// TIA Portal V17 export
// export: Created 2023-09-11T16:36:44.884775Z, ExportSetting WithDefaults, DisplayName Totally Integrated Automation Portal, DisplayVersion V17 Update 6, DisplayName TIA Portal Openness, DisplayVersion V17 Update 6, DisplayName TIA Portal Teamcenter Gateway, DisplayVersion V17 Update 6, DisplayName TIA Portal Version Control Interface, DisplayVersion V17, DisplayName Simotion SCOUT TIA, DisplayVersion 5.4.3.0, DisplayName TIA Portal Test Suite Advanced, DisplayVersion V17 Update 1, DisplayName SIMOCODE ES, DisplayVersion V17 Update 5, DisplayName SINAMICS Startdrive Advanced, DisplayVersion V17 SP1, DisplayName SINAMICS Startdrive G130, G150, S120, S150, SINAMICS MV, S210, DisplayVersion V17 SP1, DisplayName SINAMICS Startdrive G110M, G120, G120C, G120D, G120P, G115D, DisplayVersion V17 SP1, DisplayName SIRIUS Safety ES, DisplayVersion V17 Update 5, DisplayName STEP 7 Professional, DisplayVersion V17 Update 6, DisplayName STEP 7 CFC, DisplayVersion V17 Update 1, DisplayName STEP 7 Safety, DisplayVersion V17 Update 6, DisplayName WinCC Advanced, DisplayVersion V17 Update 6, DisplayName SIMATIC Visualization Architect, DisplayVersion V17 Update 5
FUNCTION "08_Gate Manager" : Void   // FC9, F_LAD
{ S7_Optimized_Access := 'TRUE' }
VERSION : 0.1
// stored: AutoNumber true, IsIECCheckEnabled false, UDAEnableTagReadback false
   VAR_TEMP
      temp_EXAMPLE_OPEN : Bool;
   END_VAR
BEGIN

REGION Network 1: S1 - SE01-B1 ([D002] P1004 | =SC01+LV004.EL001/310)
   // Sorter Gate
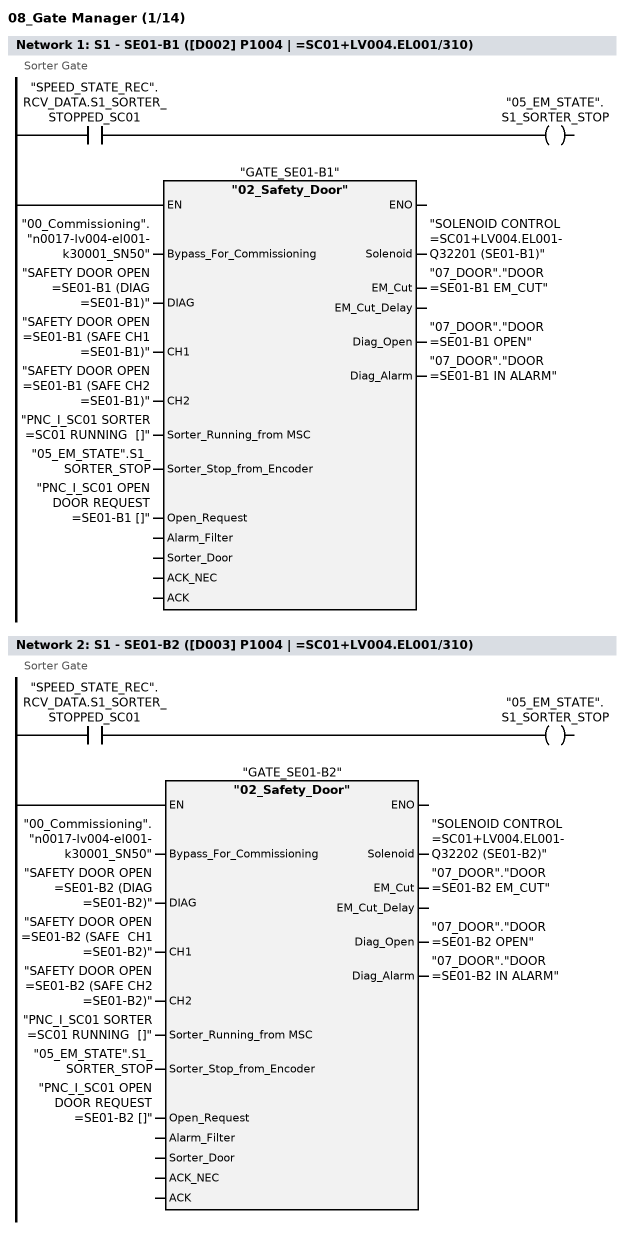
   RUNG wire#powerrail
      Contact( "SPEED_STATE_REC".RCV_DATA.S1_SORTER_STOPPED_SC01 )
      Coil( "05_EM_STATE".S1_SORTER_STOP )
   END_RUNG
   RUNG wire#powerrail
      "GATE_SE01-B1"(Bypass_For_Commissioning := "00_Commissioning"."n0017-lv004-el001-k30001_SN50", DIAG := "SAFETY DOOR OPEN =SE01-B1 (DIAG  =SE01-B1)", CH1 := "SAFETY DOOR OPEN =SE01-B1 (SAFE CH1 =SE01-B1)", CH2 := "SAFETY DOOR OPEN =SE01-B1 (SAFE CH2 =SE01-B1)", "Sorter_Running_from MSC" := "PNC_I_SC01 SORTER =SC01 RUNNING  []", Sorter_Stop_from_Encoder := "05_EM_STATE".S1_SORTER_STOP, Open_Request := "PNC_I_SC01 OPEN DOOR REQUEST =SE01-B1 []", Alarm_Filter :=, Sorter_Door :=, ACK_NEC :=, ACK :=, Solenoid => "SOLENOID CONTROL =SC01+LV004.EL001-Q32201 (SE01-B1)", EM_Cut => "07_DOOR"."DOOR =SE01-B1 EM_CUT", EM_Cut_Delay =>, Diag_Open => "07_DOOR"."DOOR =SE01-B1 OPEN", Diag_Alarm => "07_DOOR"."DOOR =SE01-B1 IN ALARM")
   END_RUNG
   // the same network as SCL:
   "05_EM_STATE".S1_SORTER_STOP := "SPEED_STATE_REC".RCV_DATA.S1_SORTER_STOPPED_SC01;
   "GATE_SE01-B1"(Bypass_For_Commissioning := "00_Commissioning"."n0017-lv004-el001-k30001_SN50",   // "02_Safety_Door"
                  DIAG := "SAFETY DOOR OPEN =SE01-B1 (DIAG  =SE01-B1)",
                  CH1 := "SAFETY DOOR OPEN =SE01-B1 (SAFE CH1 =SE01-B1)",
                  CH2 := "SAFETY DOOR OPEN =SE01-B1 (SAFE CH2 =SE01-B1)",
                  "Sorter_Running_from MSC" := "PNC_I_SC01 SORTER =SC01 RUNNING  []",
                  Sorter_Stop_from_Encoder := "05_EM_STATE".S1_SORTER_STOP,
                  Open_Request := "PNC_I_SC01 OPEN DOOR REQUEST =SE01-B1 []",
                  Solenoid => "SOLENOID CONTROL =SC01+LV004.EL001-Q32201 (SE01-B1)",
                  EM_Cut => "07_DOOR"."DOOR =SE01-B1 EM_CUT",
                  Diag_Open => "07_DOOR"."DOOR =SE01-B1 OPEN",
                  Diag_Alarm => "07_DOOR"."DOOR =SE01-B1 IN ALARM");
END_REGION

REGION Network 2: S1 - SE01-B2 ([D003] P1004 | =SC01+LV004.EL001/310)
   // Sorter Gate
   RUNG wire#powerrail
      Contact( "SPEED_STATE_REC".RCV_DATA.S1_SORTER_STOPPED_SC01 )
      Coil( "05_EM_STATE".S1_SORTER_STOP )
   END_RUNG
   RUNG wire#powerrail
      "GATE_SE01-B2"(Bypass_For_Commissioning := "00_Commissioning"."n0017-lv004-el001-k30001_SN50", DIAG := "SAFETY DOOR OPEN =SE01-B2 (DIAG  =SE01-B2)", CH1 := "SAFETY DOOR OPEN =SE01-B2 (SAFE  CH1 =SE01-B2)", CH2 := "SAFETY DOOR OPEN =SE01-B2 (SAFE CH2 =SE01-B2)", "Sorter_Running_from MSC" := "PNC_I_SC01 SORTER =SC01 RUNNING  []", Sorter_Stop_from_Encoder := "05_EM_STATE".S1_SORTER_STOP, Open_Request := "PNC_I_SC01 OPEN DOOR REQUEST =SE01-B2 []", Alarm_Filter :=, Sorter_Door :=, ACK_NEC :=, ACK :=, Solenoid => "SOLENOID CONTROL =SC01+LV004.EL001-Q32202 (SE01-B2)", EM_Cut => "07_DOOR"."DOOR =SE01-B2 EM_CUT", EM_Cut_Delay =>, Diag_Open => "07_DOOR"."DOOR =SE01-B2 OPEN", Diag_Alarm => "07_DOOR"."DOOR =SE01-B2 IN ALARM")
   END_RUNG
   // the same network as SCL:
   "05_EM_STATE".S1_SORTER_STOP := "SPEED_STATE_REC".RCV_DATA.S1_SORTER_STOPPED_SC01;
   "GATE_SE01-B2"(Bypass_For_Commissioning := "00_Commissioning"."n0017-lv004-el001-k30001_SN50",   // "02_Safety_Door"
                  DIAG := "SAFETY DOOR OPEN =SE01-B2 (DIAG  =SE01-B2)",
                  CH1 := "SAFETY DOOR OPEN =SE01-B2 (SAFE  CH1 =SE01-B2)",
                  CH2 := "SAFETY DOOR OPEN =SE01-B2 (SAFE CH2 =SE01-B2)",
                  "Sorter_Running_from MSC" := "PNC_I_SC01 SORTER =SC01 RUNNING  []",
                  Sorter_Stop_from_Encoder := "05_EM_STATE".S1_SORTER_STOP,
                  Open_Request := "PNC_I_SC01 OPEN DOOR REQUEST =SE01-B2 []",
                  Solenoid => "SOLENOID CONTROL =SC01+LV004.EL001-Q32202 (SE01-B2)",
                  EM_Cut => "07_DOOR"."DOOR =SE01-B2 EM_CUT",
                  Diag_Open => "07_DOOR"."DOOR =SE01-B2 OPEN",
                  Diag_Alarm => "07_DOOR"."DOOR =SE01-B2 IN ALARM");
END_REGION

REGION Network 3: S1 - SE01-B3 ([D012] F1001 | =SC01+MA001.EL001/310)
   // Sorter Gate
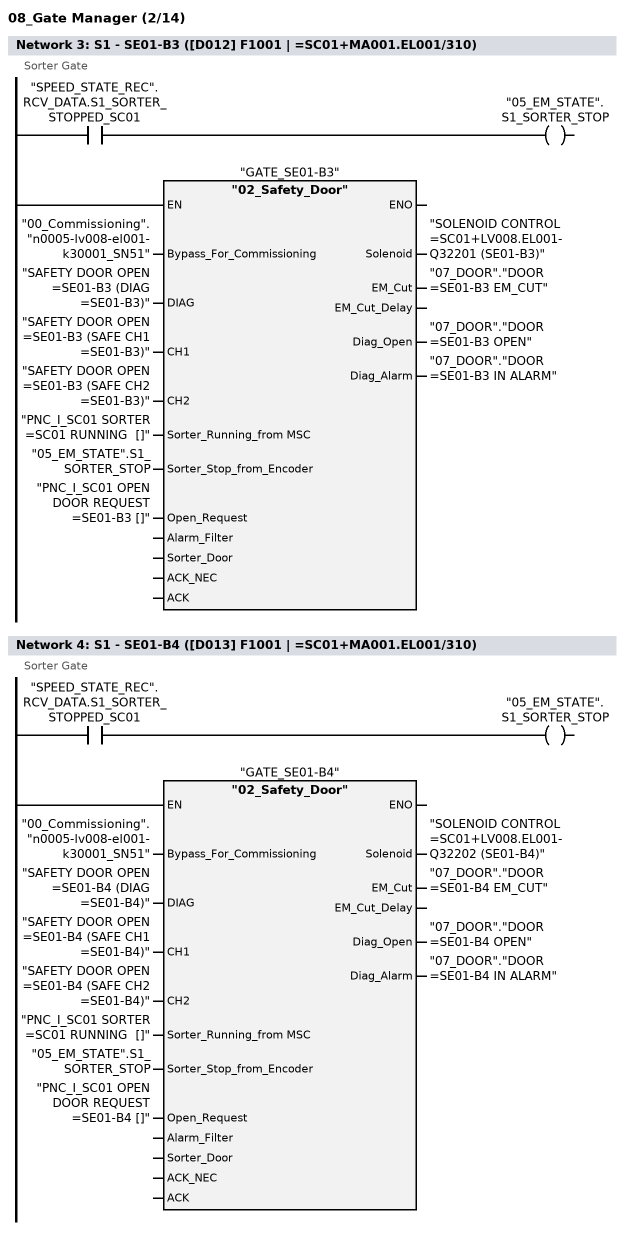
   RUNG wire#powerrail
      Contact( "SPEED_STATE_REC".RCV_DATA.S1_SORTER_STOPPED_SC01 )
      Coil( "05_EM_STATE".S1_SORTER_STOP )
   END_RUNG
   RUNG wire#powerrail
      "GATE_SE01-B3"(Bypass_For_Commissioning := "00_Commissioning"."n0005-lv008-el001-k30001_SN51", DIAG := "SAFETY DOOR OPEN =SE01-B3 (DIAG =SE01-B3)", CH1 := "SAFETY DOOR OPEN =SE01-B3 (SAFE CH1 =SE01-B3)", CH2 := "SAFETY DOOR OPEN =SE01-B3 (SAFE CH2 =SE01-B3)", "Sorter_Running_from MSC" := "PNC_I_SC01 SORTER =SC01 RUNNING  []", Sorter_Stop_from_Encoder := "05_EM_STATE".S1_SORTER_STOP, Open_Request := "PNC_I_SC01 OPEN DOOR REQUEST =SE01-B3 []", Alarm_Filter :=, Sorter_Door :=, ACK_NEC :=, ACK :=, Solenoid => "SOLENOID CONTROL =SC01+LV008.EL001-Q32201 (SE01-B3)", EM_Cut => "07_DOOR"."DOOR =SE01-B3 EM_CUT", EM_Cut_Delay =>, Diag_Open => "07_DOOR"."DOOR =SE01-B3 OPEN", Diag_Alarm => "07_DOOR"."DOOR =SE01-B3 IN ALARM")
   END_RUNG
   // the same network as SCL:
   "05_EM_STATE".S1_SORTER_STOP := "SPEED_STATE_REC".RCV_DATA.S1_SORTER_STOPPED_SC01;
   "GATE_SE01-B3"(Bypass_For_Commissioning := "00_Commissioning"."n0005-lv008-el001-k30001_SN51",   // "02_Safety_Door"
                  DIAG := "SAFETY DOOR OPEN =SE01-B3 (DIAG =SE01-B3)",
                  CH1 := "SAFETY DOOR OPEN =SE01-B3 (SAFE CH1 =SE01-B3)",
                  CH2 := "SAFETY DOOR OPEN =SE01-B3 (SAFE CH2 =SE01-B3)",
                  "Sorter_Running_from MSC" := "PNC_I_SC01 SORTER =SC01 RUNNING  []",
                  Sorter_Stop_from_Encoder := "05_EM_STATE".S1_SORTER_STOP,
                  Open_Request := "PNC_I_SC01 OPEN DOOR REQUEST =SE01-B3 []",
                  Solenoid => "SOLENOID CONTROL =SC01+LV008.EL001-Q32201 (SE01-B3)",
                  EM_Cut => "07_DOOR"."DOOR =SE01-B3 EM_CUT",
                  Diag_Open => "07_DOOR"."DOOR =SE01-B3 OPEN",
                  Diag_Alarm => "07_DOOR"."DOOR =SE01-B3 IN ALARM");
END_REGION

REGION Network 4: S1 - SE01-B4 ([D013] F1001 | =SC01+MA001.EL001/310)
   // Sorter Gate
   RUNG wire#powerrail
      Contact( "SPEED_STATE_REC".RCV_DATA.S1_SORTER_STOPPED_SC01 )
      Coil( "05_EM_STATE".S1_SORTER_STOP )
   END_RUNG
   RUNG wire#powerrail
      "GATE_SE01-B4"(Bypass_For_Commissioning := "00_Commissioning"."n0005-lv008-el001-k30001_SN51", DIAG := "SAFETY DOOR OPEN =SE01-B4 (DIAG =SE01-B4)", CH1 := "SAFETY DOOR OPEN =SE01-B4 (SAFE CH1 =SE01-B4)", CH2 := "SAFETY DOOR OPEN =SE01-B4 (SAFE CH2 =SE01-B4)", "Sorter_Running_from MSC" := "PNC_I_SC01 SORTER =SC01 RUNNING  []", Sorter_Stop_from_Encoder := "05_EM_STATE".S1_SORTER_STOP, Open_Request := "PNC_I_SC01 OPEN DOOR REQUEST =SE01-B4 []", Alarm_Filter :=, Sorter_Door :=, ACK_NEC :=, ACK :=, Solenoid => "SOLENOID CONTROL =SC01+LV008.EL001-Q32202 (SE01-B4)", EM_Cut => "07_DOOR"."DOOR =SE01-B4 EM_CUT", EM_Cut_Delay =>, Diag_Open => "07_DOOR"."DOOR =SE01-B4 OPEN", Diag_Alarm => "07_DOOR"."DOOR =SE01-B4 IN ALARM")
   END_RUNG
   // the same network as SCL:
   "05_EM_STATE".S1_SORTER_STOP := "SPEED_STATE_REC".RCV_DATA.S1_SORTER_STOPPED_SC01;
   "GATE_SE01-B4"(Bypass_For_Commissioning := "00_Commissioning"."n0005-lv008-el001-k30001_SN51",   // "02_Safety_Door"
                  DIAG := "SAFETY DOOR OPEN =SE01-B4 (DIAG =SE01-B4)",
                  CH1 := "SAFETY DOOR OPEN =SE01-B4 (SAFE CH1 =SE01-B4)",
                  CH2 := "SAFETY DOOR OPEN =SE01-B4 (SAFE CH2 =SE01-B4)",
                  "Sorter_Running_from MSC" := "PNC_I_SC01 SORTER =SC01 RUNNING  []",
                  Sorter_Stop_from_Encoder := "05_EM_STATE".S1_SORTER_STOP,
                  Open_Request := "PNC_I_SC01 OPEN DOOR REQUEST =SE01-B4 []",
                  Solenoid => "SOLENOID CONTROL =SC01+LV008.EL001-Q32202 (SE01-B4)",
                  EM_Cut => "07_DOOR"."DOOR =SE01-B4 EM_CUT",
                  Diag_Open => "07_DOOR"."DOOR =SE01-B4 OPEN",
                  Diag_Alarm => "07_DOOR"."DOOR =SE01-B4 IN ALARM");
END_REGION

REGION Network 5: S2 - SE01-B5 ([D004] P1012 | =SC02+LV004.EL001/310)
   // Sorter Gate
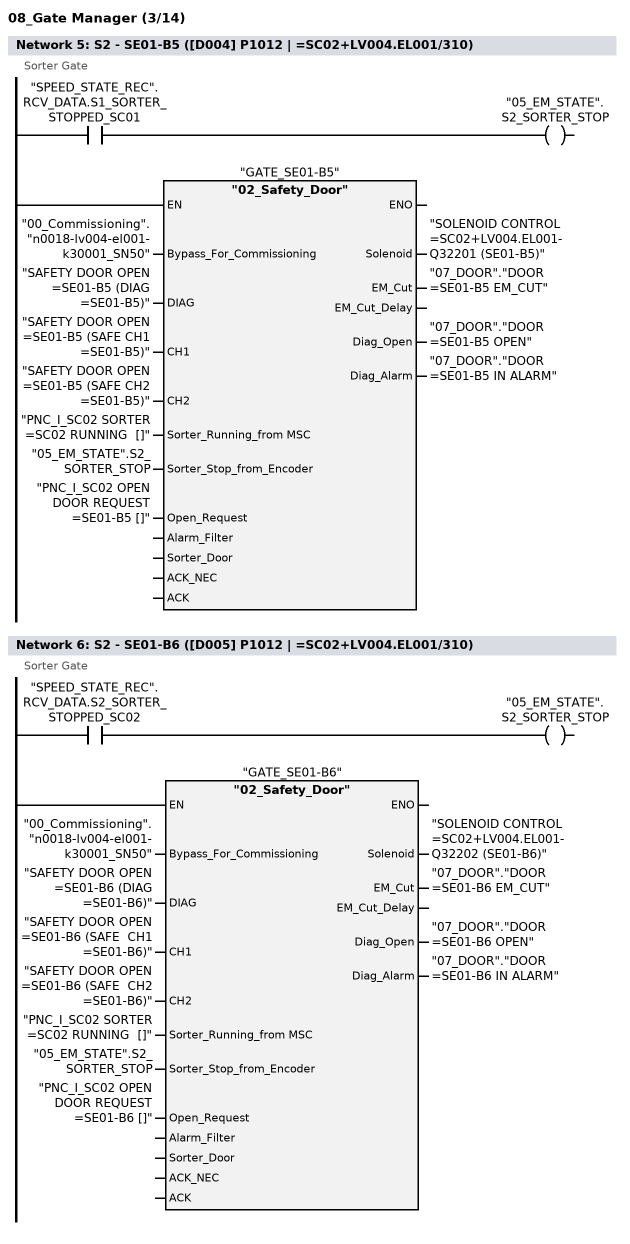
   RUNG wire#powerrail
      Contact( "SPEED_STATE_REC".RCV_DATA.S1_SORTER_STOPPED_SC01 )
      Coil( "05_EM_STATE".S2_SORTER_STOP )
   END_RUNG
   RUNG wire#powerrail
      "GATE_SE01-B5"(Bypass_For_Commissioning := "00_Commissioning"."n0018-lv004-el001-k30001_SN50", DIAG := "SAFETY DOOR OPEN =SE01-B5 (DIAG =SE01-B5)", CH1 := "SAFETY DOOR OPEN =SE01-B5 (SAFE CH1 =SE01-B5)", CH2 := "SAFETY DOOR OPEN =SE01-B5 (SAFE CH2 =SE01-B5)", "Sorter_Running_from MSC" := "PNC_I_SC02 SORTER =SC02 RUNNING  []", Sorter_Stop_from_Encoder := "05_EM_STATE".S2_SORTER_STOP, Open_Request := "PNC_I_SC02 OPEN DOOR REQUEST =SE01-B5 []", Alarm_Filter :=, Sorter_Door :=, ACK_NEC :=, ACK :=, Solenoid => "SOLENOID CONTROL =SC02+LV004.EL001-Q32201 (SE01-B5)", EM_Cut => "07_DOOR"."DOOR =SE01-B5 EM_CUT", EM_Cut_Delay =>, Diag_Open => "07_DOOR"."DOOR =SE01-B5 OPEN", Diag_Alarm => "07_DOOR"."DOOR =SE01-B5 IN ALARM")
   END_RUNG
   // the same network as SCL:
   "05_EM_STATE".S2_SORTER_STOP := "SPEED_STATE_REC".RCV_DATA.S1_SORTER_STOPPED_SC01;
   "GATE_SE01-B5"(Bypass_For_Commissioning := "00_Commissioning"."n0018-lv004-el001-k30001_SN50",   // "02_Safety_Door"
                  DIAG := "SAFETY DOOR OPEN =SE01-B5 (DIAG =SE01-B5)",
                  CH1 := "SAFETY DOOR OPEN =SE01-B5 (SAFE CH1 =SE01-B5)",
                  CH2 := "SAFETY DOOR OPEN =SE01-B5 (SAFE CH2 =SE01-B5)",
                  "Sorter_Running_from MSC" := "PNC_I_SC02 SORTER =SC02 RUNNING  []",
                  Sorter_Stop_from_Encoder := "05_EM_STATE".S2_SORTER_STOP,
                  Open_Request := "PNC_I_SC02 OPEN DOOR REQUEST =SE01-B5 []",
                  Solenoid => "SOLENOID CONTROL =SC02+LV004.EL001-Q32201 (SE01-B5)",
                  EM_Cut => "07_DOOR"."DOOR =SE01-B5 EM_CUT",
                  Diag_Open => "07_DOOR"."DOOR =SE01-B5 OPEN",
                  Diag_Alarm => "07_DOOR"."DOOR =SE01-B5 IN ALARM");
END_REGION

REGION Network 6: S2 - SE01-B6 ([D005] P1012 | =SC02+LV004.EL001/310)
   // Sorter Gate
   RUNG wire#powerrail
      Contact( "SPEED_STATE_REC".RCV_DATA.S2_SORTER_STOPPED_SC02 )
      Coil( "05_EM_STATE".S2_SORTER_STOP )
   END_RUNG
   RUNG wire#powerrail
      "GATE_SE01-B6"(Bypass_For_Commissioning := "00_Commissioning"."n0018-lv004-el001-k30001_SN50", DIAG := "SAFETY DOOR OPEN =SE01-B6 (DIAG =SE01-B6)", CH1 := "SAFETY DOOR OPEN =SE01-B6 (SAFE  CH1 =SE01-B6)", CH2 := "SAFETY DOOR OPEN =SE01-B6 (SAFE  CH2 =SE01-B6)", "Sorter_Running_from MSC" := "PNC_I_SC02 SORTER =SC02 RUNNING  []", Sorter_Stop_from_Encoder := "05_EM_STATE".S2_SORTER_STOP, Open_Request := "PNC_I_SC02 OPEN DOOR REQUEST =SE01-B6 []", Alarm_Filter :=, Sorter_Door :=, ACK_NEC :=, ACK :=, Solenoid => "SOLENOID CONTROL =SC02+LV004.EL001-Q32202 (SE01-B6)", EM_Cut => "07_DOOR"."DOOR =SE01-B6 EM_CUT", EM_Cut_Delay =>, Diag_Open => "07_DOOR"."DOOR =SE01-B6 OPEN", Diag_Alarm => "07_DOOR"."DOOR =SE01-B6 IN ALARM")
   END_RUNG
   // the same network as SCL:
   "05_EM_STATE".S2_SORTER_STOP := "SPEED_STATE_REC".RCV_DATA.S2_SORTER_STOPPED_SC02;
   "GATE_SE01-B6"(Bypass_For_Commissioning := "00_Commissioning"."n0018-lv004-el001-k30001_SN50",   // "02_Safety_Door"
                  DIAG := "SAFETY DOOR OPEN =SE01-B6 (DIAG =SE01-B6)",
                  CH1 := "SAFETY DOOR OPEN =SE01-B6 (SAFE  CH1 =SE01-B6)",
                  CH2 := "SAFETY DOOR OPEN =SE01-B6 (SAFE  CH2 =SE01-B6)",
                  "Sorter_Running_from MSC" := "PNC_I_SC02 SORTER =SC02 RUNNING  []",
                  Sorter_Stop_from_Encoder := "05_EM_STATE".S2_SORTER_STOP,
                  Open_Request := "PNC_I_SC02 OPEN DOOR REQUEST =SE01-B6 []",
                  Solenoid => "SOLENOID CONTROL =SC02+LV004.EL001-Q32202 (SE01-B6)",
                  EM_Cut => "07_DOOR"."DOOR =SE01-B6 EM_CUT",
                  Diag_Open => "07_DOOR"."DOOR =SE01-B6 OPEN",
                  Diag_Alarm => "07_DOOR"."DOOR =SE01-B6 IN ALARM");
END_REGION

REGION Network 7: S2 - SE01-B7 ([D014] F1002 | =SC02+MA001.EL001/310)
   // Sorter Gate
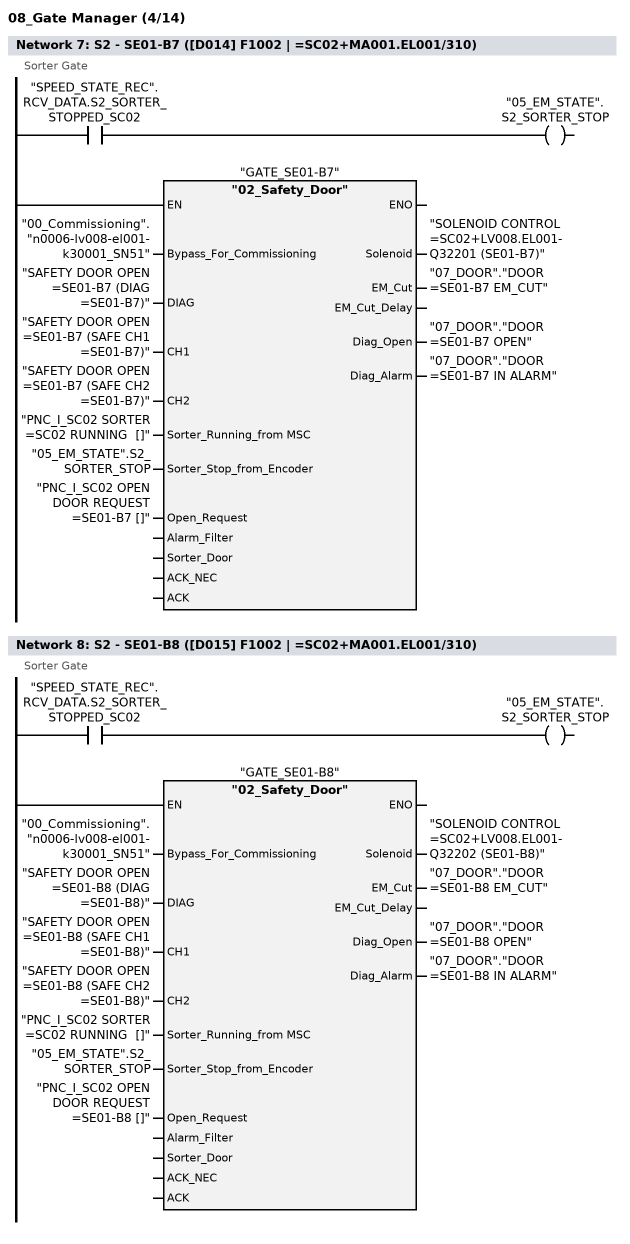
   RUNG wire#powerrail
      Contact( "SPEED_STATE_REC".RCV_DATA.S2_SORTER_STOPPED_SC02 )
      Coil( "05_EM_STATE".S2_SORTER_STOP )
   END_RUNG
   RUNG wire#powerrail
      "GATE_SE01-B7"(Bypass_For_Commissioning := "00_Commissioning"."n0006-lv008-el001-k30001_SN51", DIAG := "SAFETY DOOR OPEN =SE01-B7 (DIAG  =SE01-B7)", CH1 := "SAFETY DOOR OPEN =SE01-B7 (SAFE CH1 =SE01-B7)", CH2 := "SAFETY DOOR OPEN =SE01-B7 (SAFE CH2 =SE01-B7)", "Sorter_Running_from MSC" := "PNC_I_SC02 SORTER =SC02 RUNNING  []", Sorter_Stop_from_Encoder := "05_EM_STATE".S2_SORTER_STOP, Open_Request := "PNC_I_SC02 OPEN DOOR REQUEST =SE01-B7 []", Alarm_Filter :=, Sorter_Door :=, ACK_NEC :=, ACK :=, Solenoid => "SOLENOID CONTROL =SC02+LV008.EL001-Q32201 (SE01-B7)", EM_Cut => "07_DOOR"."DOOR =SE01-B7 EM_CUT", EM_Cut_Delay =>, Diag_Open => "07_DOOR"."DOOR =SE01-B7 OPEN", Diag_Alarm => "07_DOOR"."DOOR =SE01-B7 IN ALARM")
   END_RUNG
   // the same network as SCL:
   "05_EM_STATE".S2_SORTER_STOP := "SPEED_STATE_REC".RCV_DATA.S2_SORTER_STOPPED_SC02;
   "GATE_SE01-B7"(Bypass_For_Commissioning := "00_Commissioning"."n0006-lv008-el001-k30001_SN51",   // "02_Safety_Door"
                  DIAG := "SAFETY DOOR OPEN =SE01-B7 (DIAG  =SE01-B7)",
                  CH1 := "SAFETY DOOR OPEN =SE01-B7 (SAFE CH1 =SE01-B7)",
                  CH2 := "SAFETY DOOR OPEN =SE01-B7 (SAFE CH2 =SE01-B7)",
                  "Sorter_Running_from MSC" := "PNC_I_SC02 SORTER =SC02 RUNNING  []",
                  Sorter_Stop_from_Encoder := "05_EM_STATE".S2_SORTER_STOP,
                  Open_Request := "PNC_I_SC02 OPEN DOOR REQUEST =SE01-B7 []",
                  Solenoid => "SOLENOID CONTROL =SC02+LV008.EL001-Q32201 (SE01-B7)",
                  EM_Cut => "07_DOOR"."DOOR =SE01-B7 EM_CUT",
                  Diag_Open => "07_DOOR"."DOOR =SE01-B7 OPEN",
                  Diag_Alarm => "07_DOOR"."DOOR =SE01-B7 IN ALARM");
END_REGION

REGION Network 8: S2 - SE01-B8 ([D015] F1002 | =SC02+MA001.EL001/310)
   // Sorter Gate
   RUNG wire#powerrail
      Contact( "SPEED_STATE_REC".RCV_DATA.S2_SORTER_STOPPED_SC02 )
      Coil( "05_EM_STATE".S2_SORTER_STOP )
   END_RUNG
   RUNG wire#powerrail
      "GATE_SE01-B8"(Bypass_For_Commissioning := "00_Commissioning"."n0006-lv008-el001-k30001_SN51", DIAG := "SAFETY DOOR OPEN =SE01-B8 (DIAG  =SE01-B8)", CH1 := "SAFETY DOOR OPEN =SE01-B8 (SAFE CH1 =SE01-B8)", CH2 := "SAFETY DOOR OPEN =SE01-B8 (SAFE CH2 =SE01-B8)", "Sorter_Running_from MSC" := "PNC_I_SC02 SORTER =SC02 RUNNING  []", Sorter_Stop_from_Encoder := "05_EM_STATE".S2_SORTER_STOP, Open_Request := "PNC_I_SC02 OPEN DOOR REQUEST =SE01-B8 []", Alarm_Filter :=, Sorter_Door :=, ACK_NEC :=, ACK :=, Solenoid => "SOLENOID CONTROL =SC02+LV008.EL001-Q32202 (SE01-B8)", EM_Cut => "07_DOOR"."DOOR =SE01-B8 EM_CUT", EM_Cut_Delay =>, Diag_Open => "07_DOOR"."DOOR =SE01-B8 OPEN", Diag_Alarm => "07_DOOR"."DOOR =SE01-B8 IN ALARM")
   END_RUNG
   // the same network as SCL:
   "05_EM_STATE".S2_SORTER_STOP := "SPEED_STATE_REC".RCV_DATA.S2_SORTER_STOPPED_SC02;
   "GATE_SE01-B8"(Bypass_For_Commissioning := "00_Commissioning"."n0006-lv008-el001-k30001_SN51",   // "02_Safety_Door"
                  DIAG := "SAFETY DOOR OPEN =SE01-B8 (DIAG  =SE01-B8)",
                  CH1 := "SAFETY DOOR OPEN =SE01-B8 (SAFE CH1 =SE01-B8)",
                  CH2 := "SAFETY DOOR OPEN =SE01-B8 (SAFE CH2 =SE01-B8)",
                  "Sorter_Running_from MSC" := "PNC_I_SC02 SORTER =SC02 RUNNING  []",
                  Sorter_Stop_from_Encoder := "05_EM_STATE".S2_SORTER_STOP,
                  Open_Request := "PNC_I_SC02 OPEN DOOR REQUEST =SE01-B8 []",
                  Solenoid => "SOLENOID CONTROL =SC02+LV008.EL001-Q32202 (SE01-B8)",
                  EM_Cut => "07_DOOR"."DOOR =SE01-B8 EM_CUT",
                  Diag_Open => "07_DOOR"."DOOR =SE01-B8 OPEN",
                  Diag_Alarm => "07_DOOR"."DOOR =SE01-B8 IN ALARM");
END_REGION

REGION Network 9: S3 - SE01-B9 ([D024] F1003 | =SF03+MA001.EL001/310)
   // Sorter Gate
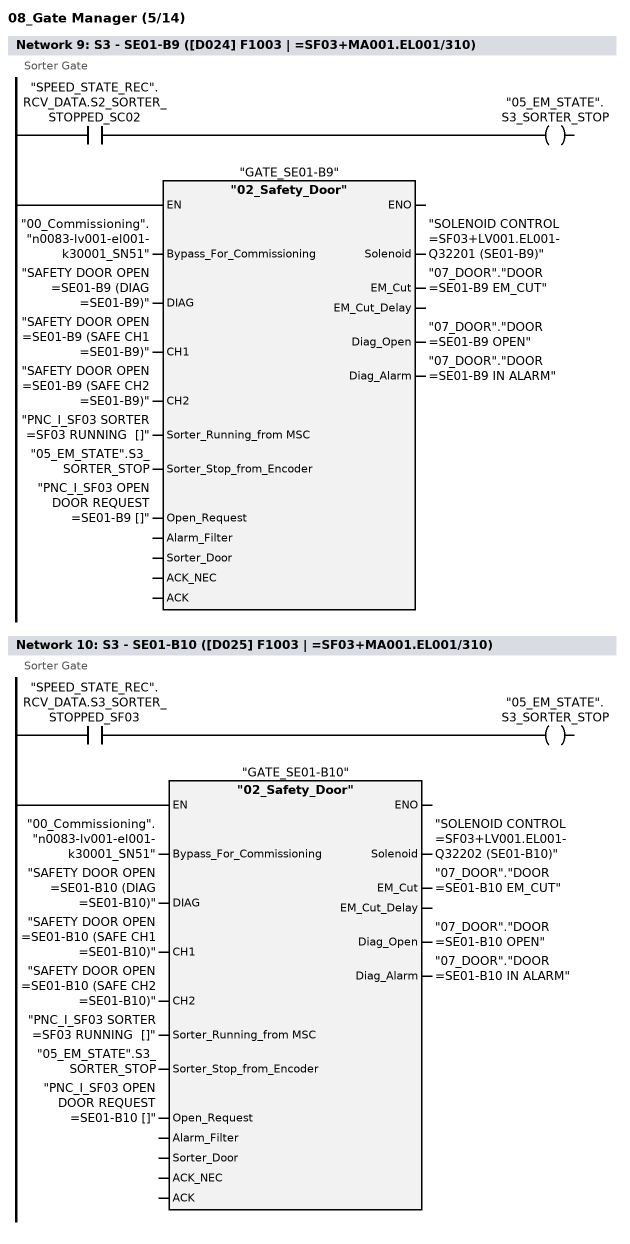
   RUNG wire#powerrail
      Contact( "SPEED_STATE_REC".RCV_DATA.S2_SORTER_STOPPED_SC02 )
      Coil( "05_EM_STATE".S3_SORTER_STOP )
   END_RUNG
   RUNG wire#powerrail
      "GATE_SE01-B9"(Bypass_For_Commissioning := "00_Commissioning"."n0083-lv001-el001-k30001_SN51", DIAG := "SAFETY DOOR OPEN =SE01-B9 (DIAG =SE01-B9)", CH1 := "SAFETY DOOR OPEN =SE01-B9 (SAFE CH1 =SE01-B9)", CH2 := "SAFETY DOOR OPEN =SE01-B9 (SAFE CH2 =SE01-B9)", "Sorter_Running_from MSC" := "PNC_I_SF03 SORTER =SF03 RUNNING  []", Sorter_Stop_from_Encoder := "05_EM_STATE".S3_SORTER_STOP, Open_Request := "PNC_I_SF03 OPEN DOOR REQUEST =SE01-B9 []", Alarm_Filter :=, Sorter_Door :=, ACK_NEC :=, ACK :=, Solenoid => "SOLENOID CONTROL =SF03+LV001.EL001-Q32201 (SE01-B9)", EM_Cut => "07_DOOR"."DOOR =SE01-B9 EM_CUT", EM_Cut_Delay =>, Diag_Open => "07_DOOR"."DOOR =SE01-B9 OPEN", Diag_Alarm => "07_DOOR"."DOOR =SE01-B9 IN ALARM")
   END_RUNG
   // the same network as SCL:
   "05_EM_STATE".S3_SORTER_STOP := "SPEED_STATE_REC".RCV_DATA.S2_SORTER_STOPPED_SC02;
   "GATE_SE01-B9"(Bypass_For_Commissioning := "00_Commissioning"."n0083-lv001-el001-k30001_SN51",   // "02_Safety_Door"
                  DIAG := "SAFETY DOOR OPEN =SE01-B9 (DIAG =SE01-B9)",
                  CH1 := "SAFETY DOOR OPEN =SE01-B9 (SAFE CH1 =SE01-B9)",
                  CH2 := "SAFETY DOOR OPEN =SE01-B9 (SAFE CH2 =SE01-B9)",
                  "Sorter_Running_from MSC" := "PNC_I_SF03 SORTER =SF03 RUNNING  []",
                  Sorter_Stop_from_Encoder := "05_EM_STATE".S3_SORTER_STOP,
                  Open_Request := "PNC_I_SF03 OPEN DOOR REQUEST =SE01-B9 []",
                  Solenoid => "SOLENOID CONTROL =SF03+LV001.EL001-Q32201 (SE01-B9)",
                  EM_Cut => "07_DOOR"."DOOR =SE01-B9 EM_CUT",
                  Diag_Open => "07_DOOR"."DOOR =SE01-B9 OPEN",
                  Diag_Alarm => "07_DOOR"."DOOR =SE01-B9 IN ALARM");
END_REGION

REGION Network 10: S3 - SE01-B10 ([D025] F1003 | =SF03+MA001.EL001/310)
   // Sorter Gate
   RUNG wire#powerrail
      Contact( "SPEED_STATE_REC".RCV_DATA.S3_SORTER_STOPPED_SF03 )
      Coil( "05_EM_STATE".S3_SORTER_STOP )
   END_RUNG
   RUNG wire#powerrail
      "GATE_SE01-B10"(Bypass_For_Commissioning := "00_Commissioning"."n0083-lv001-el001-k30001_SN51", DIAG := "SAFETY DOOR OPEN =SE01-B10 (DIAG =SE01-B10)", CH1 := "SAFETY DOOR OPEN =SE01-B10 (SAFE CH1 =SE01-B10)", CH2 := "SAFETY DOOR OPEN =SE01-B10 (SAFE CH2 =SE01-B10)", "Sorter_Running_from MSC" := "PNC_I_SF03 SORTER =SF03 RUNNING  []", Sorter_Stop_from_Encoder := "05_EM_STATE".S3_SORTER_STOP, Open_Request := "PNC_I_SF03 OPEN DOOR REQUEST =SE01-B10 []", Alarm_Filter :=, Sorter_Door :=, ACK_NEC :=, ACK :=, Solenoid => "SOLENOID CONTROL =SF03+LV001.EL001-Q32202 (SE01-B10)", EM_Cut => "07_DOOR"."DOOR =SE01-B10 EM_CUT", EM_Cut_Delay =>, Diag_Open => "07_DOOR"."DOOR =SE01-B10 OPEN", Diag_Alarm => "07_DOOR"."DOOR =SE01-B10 IN ALARM")
   END_RUNG
   // the same network as SCL:
   "05_EM_STATE".S3_SORTER_STOP := "SPEED_STATE_REC".RCV_DATA.S3_SORTER_STOPPED_SF03;
   "GATE_SE01-B10"(Bypass_For_Commissioning := "00_Commissioning"."n0083-lv001-el001-k30001_SN51",   // "02_Safety_Door"
                   DIAG := "SAFETY DOOR OPEN =SE01-B10 (DIAG =SE01-B10)",
                   CH1 := "SAFETY DOOR OPEN =SE01-B10 (SAFE CH1 =SE01-B10)",
                   CH2 := "SAFETY DOOR OPEN =SE01-B10 (SAFE CH2 =SE01-B10)",
                   "Sorter_Running_from MSC" := "PNC_I_SF03 SORTER =SF03 RUNNING  []",
                   Sorter_Stop_from_Encoder := "05_EM_STATE".S3_SORTER_STOP,
                   Open_Request := "PNC_I_SF03 OPEN DOOR REQUEST =SE01-B10 []",
                   Solenoid => "SOLENOID CONTROL =SF03+LV001.EL001-Q32202 (SE01-B10)",
                   EM_Cut => "07_DOOR"."DOOR =SE01-B10 EM_CUT",
                   Diag_Open => "07_DOOR"."DOOR =SE01-B10 OPEN",
                   Diag_Alarm => "07_DOOR"."DOOR =SE01-B10 IN ALARM");
END_REGION

REGION Network 11: S4 - SE01-B11 ([D026] F1004 | =SF04+MA001.EL001/310)
   // Sorter Gate
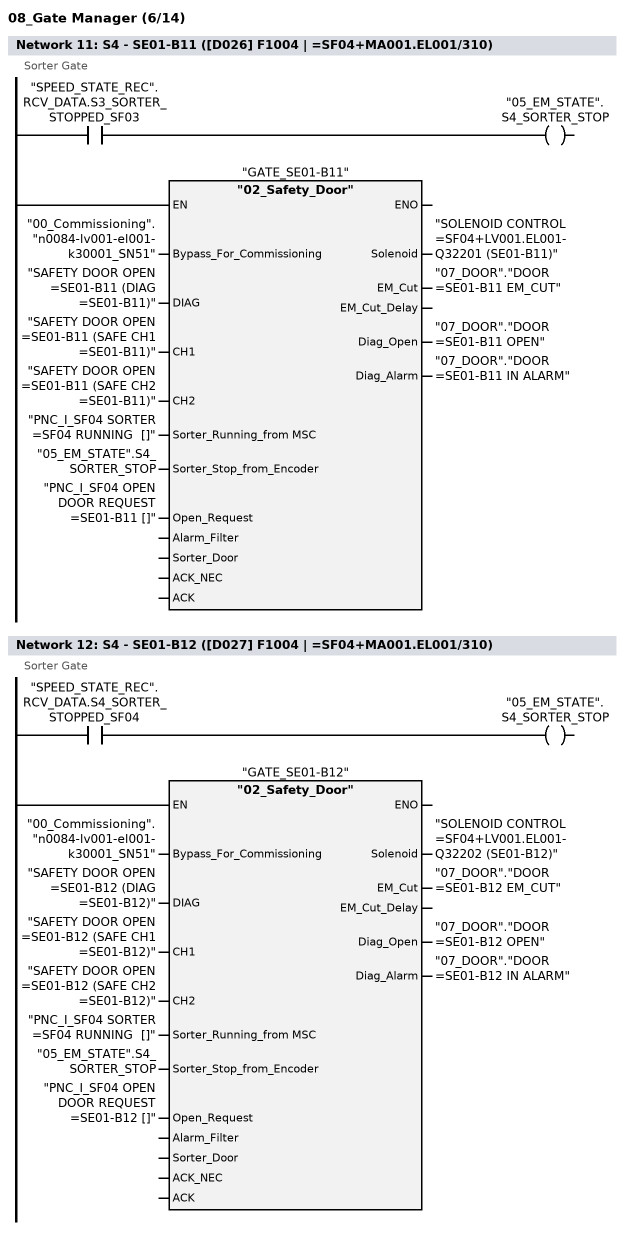
   RUNG wire#powerrail
      Contact( "SPEED_STATE_REC".RCV_DATA.S3_SORTER_STOPPED_SF03 )
      Coil( "05_EM_STATE".S4_SORTER_STOP )
   END_RUNG
   RUNG wire#powerrail
      "GATE_SE01-B11"(Bypass_For_Commissioning := "00_Commissioning"."n0084-lv001-el001-k30001_SN51", DIAG := "SAFETY DOOR OPEN =SE01-B11 (DIAG =SE01-B11)", CH1 := "SAFETY DOOR OPEN =SE01-B11 (SAFE CH1 =SE01-B11)", CH2 := "SAFETY DOOR OPEN =SE01-B11 (SAFE CH2 =SE01-B11)", "Sorter_Running_from MSC" := "PNC_I_SF04 SORTER =SF04 RUNNING  []", Sorter_Stop_from_Encoder := "05_EM_STATE".S4_SORTER_STOP, Open_Request := "PNC_I_SF04 OPEN DOOR REQUEST =SE01-B11 []", Alarm_Filter :=, Sorter_Door :=, ACK_NEC :=, ACK :=, Solenoid => "SOLENOID CONTROL =SF04+LV001.EL001-Q32201 (SE01-B11)", EM_Cut => "07_DOOR"."DOOR =SE01-B11 EM_CUT", EM_Cut_Delay =>, Diag_Open => "07_DOOR"."DOOR =SE01-B11 OPEN", Diag_Alarm => "07_DOOR"."DOOR =SE01-B11 IN ALARM")
   END_RUNG
   // the same network as SCL:
   "05_EM_STATE".S4_SORTER_STOP := "SPEED_STATE_REC".RCV_DATA.S3_SORTER_STOPPED_SF03;
   "GATE_SE01-B11"(Bypass_For_Commissioning := "00_Commissioning"."n0084-lv001-el001-k30001_SN51",   // "02_Safety_Door"
                   DIAG := "SAFETY DOOR OPEN =SE01-B11 (DIAG =SE01-B11)",
                   CH1 := "SAFETY DOOR OPEN =SE01-B11 (SAFE CH1 =SE01-B11)",
                   CH2 := "SAFETY DOOR OPEN =SE01-B11 (SAFE CH2 =SE01-B11)",
                   "Sorter_Running_from MSC" := "PNC_I_SF04 SORTER =SF04 RUNNING  []",
                   Sorter_Stop_from_Encoder := "05_EM_STATE".S4_SORTER_STOP,
                   Open_Request := "PNC_I_SF04 OPEN DOOR REQUEST =SE01-B11 []",
                   Solenoid => "SOLENOID CONTROL =SF04+LV001.EL001-Q32201 (SE01-B11)",
                   EM_Cut => "07_DOOR"."DOOR =SE01-B11 EM_CUT",
                   Diag_Open => "07_DOOR"."DOOR =SE01-B11 OPEN",
                   Diag_Alarm => "07_DOOR"."DOOR =SE01-B11 IN ALARM");
END_REGION

REGION Network 12: S4 - SE01-B12 ([D027] F1004 | =SF04+MA001.EL001/310)
   // Sorter Gate
   RUNG wire#powerrail
      Contact( "SPEED_STATE_REC".RCV_DATA.S4_SORTER_STOPPED_SF04 )
      Coil( "05_EM_STATE".S4_SORTER_STOP )
   END_RUNG
   RUNG wire#powerrail
      "GATE_SE01-B12"(Bypass_For_Commissioning := "00_Commissioning"."n0084-lv001-el001-k30001_SN51", DIAG := "SAFETY DOOR OPEN =SE01-B12 (DIAG =SE01-B12)", CH1 := "SAFETY DOOR OPEN =SE01-B12 (SAFE CH1 =SE01-B12)", CH2 := "SAFETY DOOR OPEN =SE01-B12 (SAFE CH2 =SE01-B12)", "Sorter_Running_from MSC" := "PNC_I_SF04 SORTER =SF04 RUNNING  []", Sorter_Stop_from_Encoder := "05_EM_STATE".S4_SORTER_STOP, Open_Request := "PNC_I_SF04 OPEN DOOR REQUEST =SE01-B12 []", Alarm_Filter :=, Sorter_Door :=, ACK_NEC :=, ACK :=, Solenoid => "SOLENOID CONTROL =SF04+LV001.EL001-Q32202 (SE01-B12)", EM_Cut => "07_DOOR"."DOOR =SE01-B12 EM_CUT", EM_Cut_Delay =>, Diag_Open => "07_DOOR"."DOOR =SE01-B12 OPEN", Diag_Alarm => "07_DOOR"."DOOR =SE01-B12 IN ALARM")
   END_RUNG
   // the same network as SCL:
   "05_EM_STATE".S4_SORTER_STOP := "SPEED_STATE_REC".RCV_DATA.S4_SORTER_STOPPED_SF04;
   "GATE_SE01-B12"(Bypass_For_Commissioning := "00_Commissioning"."n0084-lv001-el001-k30001_SN51",   // "02_Safety_Door"
                   DIAG := "SAFETY DOOR OPEN =SE01-B12 (DIAG =SE01-B12)",
                   CH1 := "SAFETY DOOR OPEN =SE01-B12 (SAFE CH1 =SE01-B12)",
                   CH2 := "SAFETY DOOR OPEN =SE01-B12 (SAFE CH2 =SE01-B12)",
                   "Sorter_Running_from MSC" := "PNC_I_SF04 SORTER =SF04 RUNNING  []",
                   Sorter_Stop_from_Encoder := "05_EM_STATE".S4_SORTER_STOP,
                   Open_Request := "PNC_I_SF04 OPEN DOOR REQUEST =SE01-B12 []",
                   Solenoid => "SOLENOID CONTROL =SF04+LV001.EL001-Q32202 (SE01-B12)",
                   EM_Cut => "07_DOOR"."DOOR =SE01-B12 EM_CUT",
                   Diag_Open => "07_DOOR"."DOOR =SE01-B12 OPEN",
                   Diag_Alarm => "07_DOOR"."DOOR =SE01-B12 IN ALARM");
END_REGION

REGION Network 13: L1 - SC00+UC114.VS019 ([D010] S4001 | =SC00+UC11.EL001/311)
   // Sorter Gate
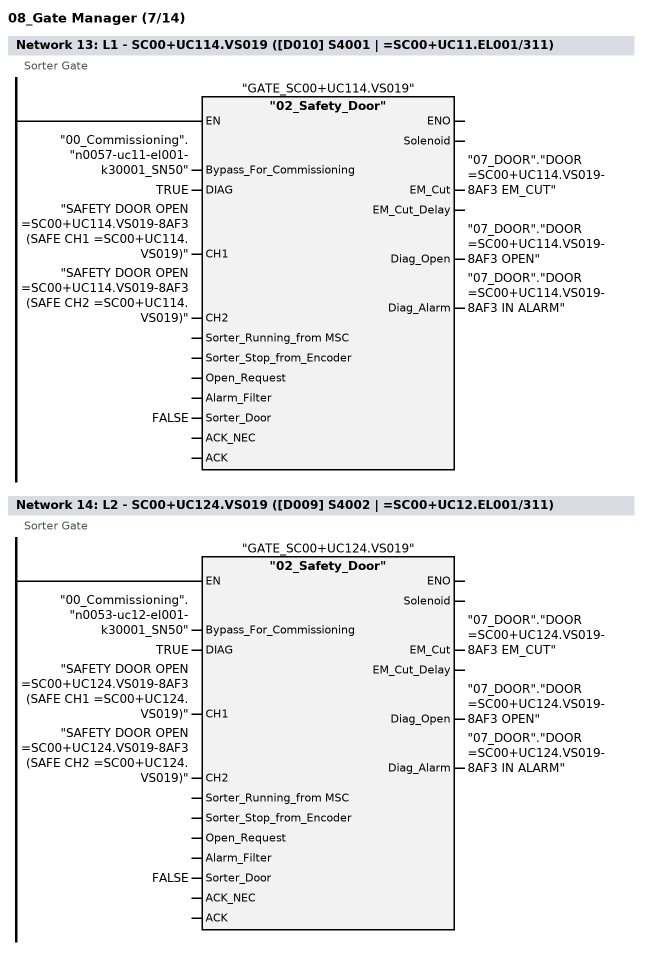
   RUNG wire#powerrail
      "GATE_SC00+UC114.VS019"(Bypass_For_Commissioning := "00_Commissioning"."n0057-uc11-el001-k30001_SN50", DIAG := TRUE, CH1 := "SAFETY DOOR OPEN =SC00+UC114.VS019-8AF3 (SAFE CH1 =SC00+UC114.VS019)", CH2 := "SAFETY DOOR OPEN =SC00+UC114.VS019-8AF3 (SAFE CH2 =SC00+UC114.VS019)", "Sorter_Running_from MSC" :=, Sorter_Stop_from_Encoder :=, Open_Request :=, Alarm_Filter :=, Sorter_Door := FALSE, ACK_NEC :=, ACK :=, Solenoid =>, EM_Cut => "07_DOOR"."DOOR =SC00+UC114.VS019-8AF3 EM_CUT", EM_Cut_Delay =>, Diag_Open => "07_DOOR"."DOOR =SC00+UC114.VS019-8AF3 OPEN", Diag_Alarm => "07_DOOR"."DOOR =SC00+UC114.VS019-8AF3 IN ALARM")
   END_RUNG
   // the same network as SCL:
   "GATE_SC00+UC114.VS019"(Bypass_For_Commissioning := "00_Commissioning"."n0057-uc11-el001-k30001_SN50",   // "02_Safety_Door"
                           DIAG := TRUE,
                           CH1 := "SAFETY DOOR OPEN =SC00+UC114.VS019-8AF3 (SAFE CH1 =SC00+UC114.VS019)",
                           CH2 := "SAFETY DOOR OPEN =SC00+UC114.VS019-8AF3 (SAFE CH2 =SC00+UC114.VS019)",
                           Sorter_Door := FALSE,
                           EM_Cut => "07_DOOR"."DOOR =SC00+UC114.VS019-8AF3 EM_CUT",
                           Diag_Open => "07_DOOR"."DOOR =SC00+UC114.VS019-8AF3 OPEN",
                           Diag_Alarm => "07_DOOR"."DOOR =SC00+UC114.VS019-8AF3 IN ALARM");
END_REGION

REGION Network 14: L2 - SC00+UC124.VS019 ([D009] S4002 | =SC00+UC12.EL001/311)
   // Sorter Gate
   RUNG wire#powerrail
      "GATE_SC00+UC124.VS019"(Bypass_For_Commissioning := "00_Commissioning"."n0053-uc12-el001-k30001_SN50", DIAG := TRUE, CH1 := "SAFETY DOOR OPEN =SC00+UC124.VS019-8AF3 (SAFE CH1 =SC00+UC124.VS019)", CH2 := "SAFETY DOOR OPEN =SC00+UC124.VS019-8AF3 (SAFE CH2 =SC00+UC124.VS019)", "Sorter_Running_from MSC" :=, Sorter_Stop_from_Encoder :=, Open_Request :=, Alarm_Filter :=, Sorter_Door := FALSE, ACK_NEC :=, ACK :=, Solenoid =>, EM_Cut => "07_DOOR"."DOOR =SC00+UC124.VS019-8AF3 EM_CUT", EM_Cut_Delay =>, Diag_Open => "07_DOOR"."DOOR =SC00+UC124.VS019-8AF3 OPEN", Diag_Alarm => "07_DOOR"."DOOR =SC00+UC124.VS019-8AF3 IN ALARM")
   END_RUNG
   // the same network as SCL:
   "GATE_SC00+UC124.VS019"(Bypass_For_Commissioning := "00_Commissioning"."n0053-uc12-el001-k30001_SN50",   // "02_Safety_Door"
                           DIAG := TRUE,
                           CH1 := "SAFETY DOOR OPEN =SC00+UC124.VS019-8AF3 (SAFE CH1 =SC00+UC124.VS019)",
                           CH2 := "SAFETY DOOR OPEN =SC00+UC124.VS019-8AF3 (SAFE CH2 =SC00+UC124.VS019)",
                           Sorter_Door := FALSE,
                           EM_Cut => "07_DOOR"."DOOR =SC00+UC124.VS019-8AF3 EM_CUT",
                           Diag_Open => "07_DOOR"."DOOR =SC00+UC124.VS019-8AF3 OPEN",
                           Diag_Alarm => "07_DOOR"."DOOR =SC00+UC124.VS019-8AF3 IN ALARM");
END_REGION

REGION Network 15: L3 - SC00+UC134.VS019 ([D008] S4003 | =SC00+UC13.EL001/311)
   // Sorter Gate
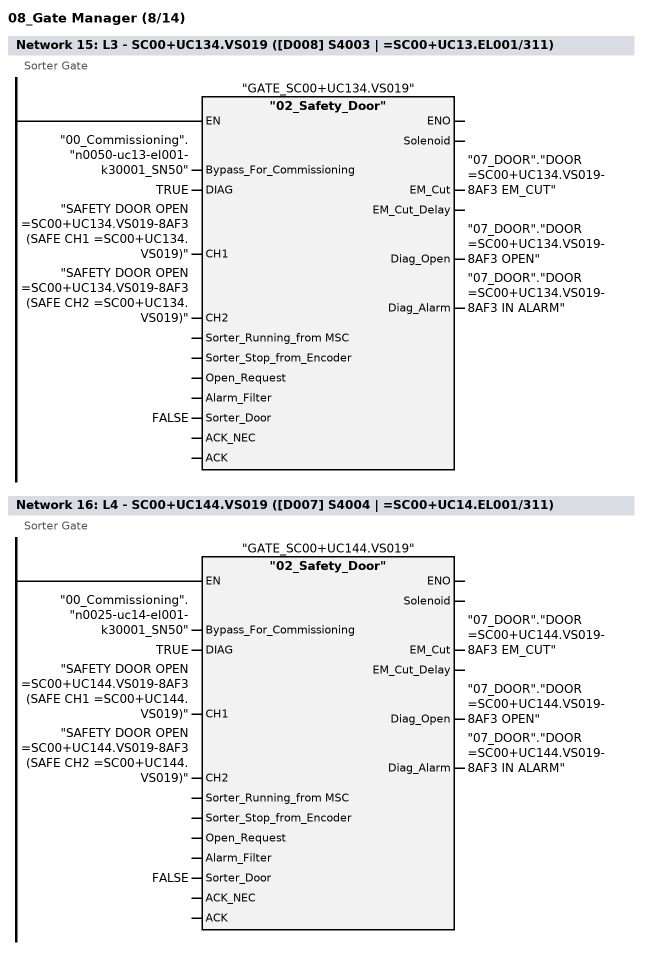
   RUNG wire#powerrail
      "GATE_SC00+UC134.VS019"(Bypass_For_Commissioning := "00_Commissioning"."n0050-uc13-el001-k30001_SN50", DIAG := TRUE, CH1 := "SAFETY DOOR OPEN =SC00+UC134.VS019-8AF3 (SAFE CH1 =SC00+UC134.VS019)", CH2 := "SAFETY DOOR OPEN =SC00+UC134.VS019-8AF3 (SAFE CH2 =SC00+UC134.VS019)", "Sorter_Running_from MSC" :=, Sorter_Stop_from_Encoder :=, Open_Request :=, Alarm_Filter :=, Sorter_Door := FALSE, ACK_NEC :=, ACK :=, Solenoid =>, EM_Cut => "07_DOOR"."DOOR =SC00+UC134.VS019-8AF3 EM_CUT", EM_Cut_Delay =>, Diag_Open => "07_DOOR"."DOOR =SC00+UC134.VS019-8AF3 OPEN", Diag_Alarm => "07_DOOR"."DOOR =SC00+UC134.VS019-8AF3 IN ALARM")
   END_RUNG
   // the same network as SCL:
   "GATE_SC00+UC134.VS019"(Bypass_For_Commissioning := "00_Commissioning"."n0050-uc13-el001-k30001_SN50",   // "02_Safety_Door"
                           DIAG := TRUE,
                           CH1 := "SAFETY DOOR OPEN =SC00+UC134.VS019-8AF3 (SAFE CH1 =SC00+UC134.VS019)",
                           CH2 := "SAFETY DOOR OPEN =SC00+UC134.VS019-8AF3 (SAFE CH2 =SC00+UC134.VS019)",
                           Sorter_Door := FALSE,
                           EM_Cut => "07_DOOR"."DOOR =SC00+UC134.VS019-8AF3 EM_CUT",
                           Diag_Open => "07_DOOR"."DOOR =SC00+UC134.VS019-8AF3 OPEN",
                           Diag_Alarm => "07_DOOR"."DOOR =SC00+UC134.VS019-8AF3 IN ALARM");
END_REGION

REGION Network 16: L4 - SC00+UC144.VS019 ([D007] S4004 | =SC00+UC14.EL001/311)
   // Sorter Gate
   RUNG wire#powerrail
      "GATE_SC00+UC144.VS019"(Bypass_For_Commissioning := "00_Commissioning"."n0025-uc14-el001-k30001_SN50", DIAG := TRUE, CH1 := "SAFETY DOOR OPEN =SC00+UC144.VS019-8AF3 (SAFE CH1 =SC00+UC144.VS019)", CH2 := "SAFETY DOOR OPEN =SC00+UC144.VS019-8AF3 (SAFE CH2 =SC00+UC144.VS019)", "Sorter_Running_from MSC" :=, Sorter_Stop_from_Encoder :=, Open_Request :=, Alarm_Filter :=, Sorter_Door := FALSE, ACK_NEC :=, ACK :=, Solenoid =>, EM_Cut => "07_DOOR"."DOOR =SC00+UC144.VS019-8AF3 EM_CUT", EM_Cut_Delay =>, Diag_Open => "07_DOOR"."DOOR =SC00+UC144.VS019-8AF3 OPEN", Diag_Alarm => "07_DOOR"."DOOR =SC00+UC144.VS019-8AF3 IN ALARM")
   END_RUNG
   // the same network as SCL:
   "GATE_SC00+UC144.VS019"(Bypass_For_Commissioning := "00_Commissioning"."n0025-uc14-el001-k30001_SN50",   // "02_Safety_Door"
                           DIAG := TRUE,
                           CH1 := "SAFETY DOOR OPEN =SC00+UC144.VS019-8AF3 (SAFE CH1 =SC00+UC144.VS019)",
                           CH2 := "SAFETY DOOR OPEN =SC00+UC144.VS019-8AF3 (SAFE CH2 =SC00+UC144.VS019)",
                           Sorter_Door := FALSE,
                           EM_Cut => "07_DOOR"."DOOR =SC00+UC144.VS019-8AF3 EM_CUT",
                           Diag_Open => "07_DOOR"."DOOR =SC00+UC144.VS019-8AF3 OPEN",
                           Diag_Alarm => "07_DOOR"."DOOR =SC00+UC144.VS019-8AF3 IN ALARM");
END_REGION

REGION Network 17: L5 - SC00+UC154.VS019 ([D006] S4005 | =SC00+UC15.EL001/311)
   // Sorter Gate
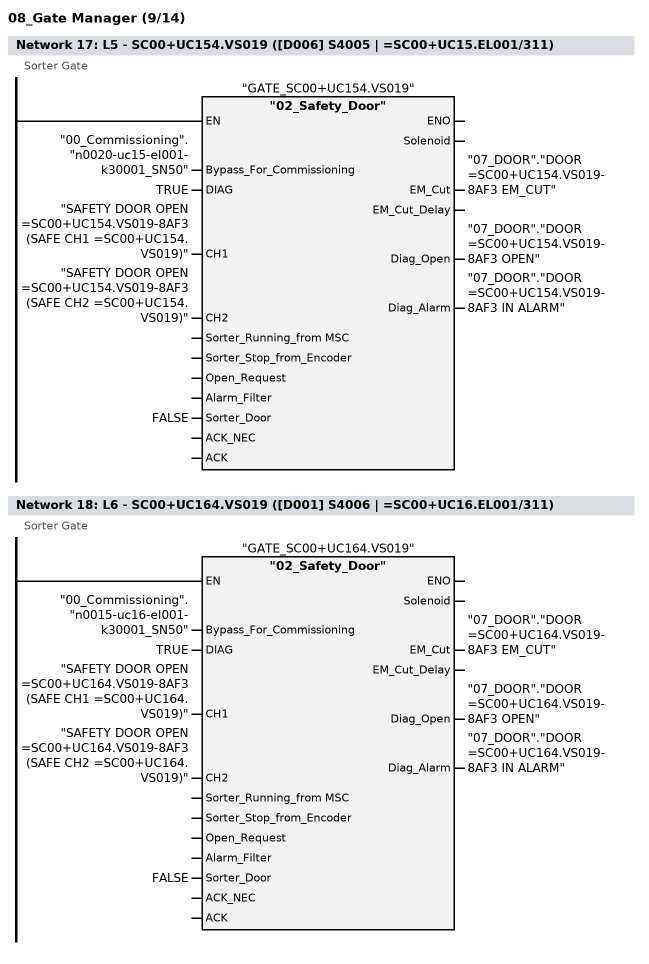
   RUNG wire#powerrail
      "GATE_SC00+UC154.VS019"(Bypass_For_Commissioning := "00_Commissioning"."n0020-uc15-el001-k30001_SN50", DIAG := TRUE, CH1 := "SAFETY DOOR OPEN =SC00+UC154.VS019-8AF3 (SAFE CH1 =SC00+UC154.VS019)", CH2 := "SAFETY DOOR OPEN =SC00+UC154.VS019-8AF3 (SAFE CH2 =SC00+UC154.VS019)", "Sorter_Running_from MSC" :=, Sorter_Stop_from_Encoder :=, Open_Request :=, Alarm_Filter :=, Sorter_Door := FALSE, ACK_NEC :=, ACK :=, Solenoid =>, EM_Cut => "07_DOOR"."DOOR =SC00+UC154.VS019-8AF3 EM_CUT", EM_Cut_Delay =>, Diag_Open => "07_DOOR"."DOOR =SC00+UC154.VS019-8AF3 OPEN", Diag_Alarm => "07_DOOR"."DOOR =SC00+UC154.VS019-8AF3 IN ALARM")
   END_RUNG
   // the same network as SCL:
   "GATE_SC00+UC154.VS019"(Bypass_For_Commissioning := "00_Commissioning"."n0020-uc15-el001-k30001_SN50",   // "02_Safety_Door"
                           DIAG := TRUE,
                           CH1 := "SAFETY DOOR OPEN =SC00+UC154.VS019-8AF3 (SAFE CH1 =SC00+UC154.VS019)",
                           CH2 := "SAFETY DOOR OPEN =SC00+UC154.VS019-8AF3 (SAFE CH2 =SC00+UC154.VS019)",
                           Sorter_Door := FALSE,
                           EM_Cut => "07_DOOR"."DOOR =SC00+UC154.VS019-8AF3 EM_CUT",
                           Diag_Open => "07_DOOR"."DOOR =SC00+UC154.VS019-8AF3 OPEN",
                           Diag_Alarm => "07_DOOR"."DOOR =SC00+UC154.VS019-8AF3 IN ALARM");
END_REGION

REGION Network 18: L6 - SC00+UC164.VS019 ([D001] S4006 | =SC00+UC16.EL001/311)
   // Sorter Gate
   RUNG wire#powerrail
      "GATE_SC00+UC164.VS019"(Bypass_For_Commissioning := "00_Commissioning"."n0015-uc16-el001-k30001_SN50", DIAG := TRUE, CH1 := "SAFETY DOOR OPEN =SC00+UC164.VS019-8AF3 (SAFE CH1 =SC00+UC164.VS019)", CH2 := "SAFETY DOOR OPEN =SC00+UC164.VS019-8AF3 (SAFE CH2 =SC00+UC164.VS019)", "Sorter_Running_from MSC" :=, Sorter_Stop_from_Encoder :=, Open_Request :=, Alarm_Filter :=, Sorter_Door := FALSE, ACK_NEC :=, ACK :=, Solenoid =>, EM_Cut => "07_DOOR"."DOOR =SC00+UC164.VS019-8AF3 EM_CUT", EM_Cut_Delay =>, Diag_Open => "07_DOOR"."DOOR =SC00+UC164.VS019-8AF3 OPEN", Diag_Alarm => "07_DOOR"."DOOR =SC00+UC164.VS019-8AF3 IN ALARM")
   END_RUNG
   // the same network as SCL:
   "GATE_SC00+UC164.VS019"(Bypass_For_Commissioning := "00_Commissioning"."n0015-uc16-el001-k30001_SN50",   // "02_Safety_Door"
                           DIAG := TRUE,
                           CH1 := "SAFETY DOOR OPEN =SC00+UC164.VS019-8AF3 (SAFE CH1 =SC00+UC164.VS019)",
                           CH2 := "SAFETY DOOR OPEN =SC00+UC164.VS019-8AF3 (SAFE CH2 =SC00+UC164.VS019)",
                           Sorter_Door := FALSE,
                           EM_Cut => "07_DOOR"."DOOR =SC00+UC164.VS019-8AF3 EM_CUT",
                           Diag_Open => "07_DOOR"."DOOR =SC00+UC164.VS019-8AF3 OPEN",
                           Diag_Alarm => "07_DOOR"."DOOR =SC00+UC164.VS019-8AF3 IN ALARM");
END_REGION

REGION Network 19: L7 - SC00+UC175.VS019 ([D011] S4007 | =SC00+UC17.EL001/310)
   // Sorter Gate
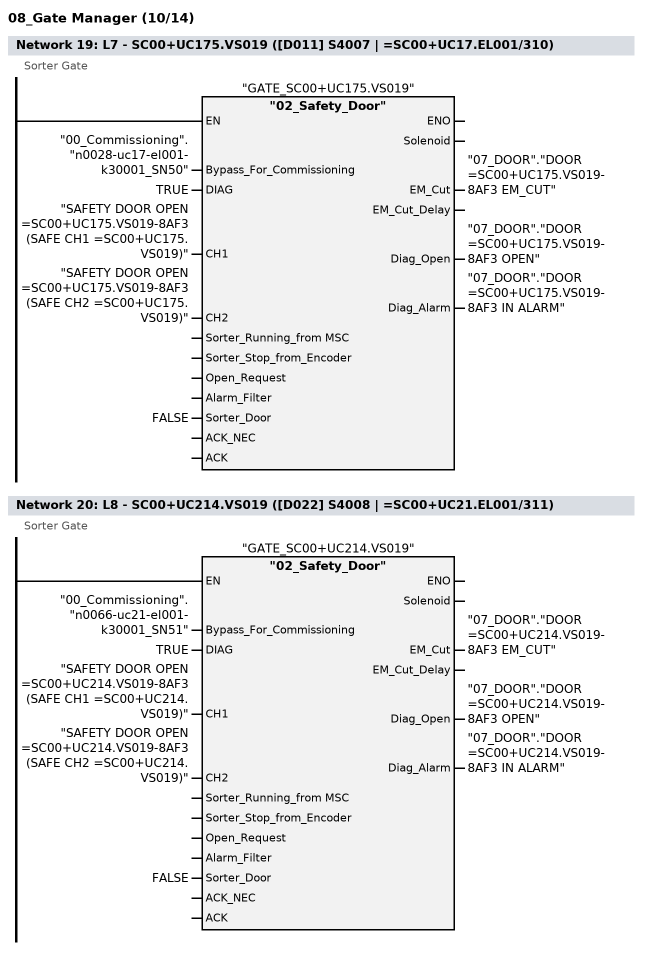
   RUNG wire#powerrail
      "GATE_SC00+UC175.VS019"(Bypass_For_Commissioning := "00_Commissioning"."n0028-uc17-el001-k30001_SN50", DIAG := TRUE, CH1 := "SAFETY DOOR OPEN =SC00+UC175.VS019-8AF3 (SAFE CH1 =SC00+UC175.VS019)", CH2 := "SAFETY DOOR OPEN =SC00+UC175.VS019-8AF3 (SAFE CH2 =SC00+UC175.VS019)", "Sorter_Running_from MSC" :=, Sorter_Stop_from_Encoder :=, Open_Request :=, Alarm_Filter :=, Sorter_Door := FALSE, ACK_NEC :=, ACK :=, Solenoid =>, EM_Cut => "07_DOOR"."DOOR =SC00+UC175.VS019-8AF3 EM_CUT", EM_Cut_Delay =>, Diag_Open => "07_DOOR"."DOOR =SC00+UC175.VS019-8AF3 OPEN", Diag_Alarm => "07_DOOR"."DOOR =SC00+UC175.VS019-8AF3 IN ALARM")
   END_RUNG
   // the same network as SCL:
   "GATE_SC00+UC175.VS019"(Bypass_For_Commissioning := "00_Commissioning"."n0028-uc17-el001-k30001_SN50",   // "02_Safety_Door"
                           DIAG := TRUE,
                           CH1 := "SAFETY DOOR OPEN =SC00+UC175.VS019-8AF3 (SAFE CH1 =SC00+UC175.VS019)",
                           CH2 := "SAFETY DOOR OPEN =SC00+UC175.VS019-8AF3 (SAFE CH2 =SC00+UC175.VS019)",
                           Sorter_Door := FALSE,
                           EM_Cut => "07_DOOR"."DOOR =SC00+UC175.VS019-8AF3 EM_CUT",
                           Diag_Open => "07_DOOR"."DOOR =SC00+UC175.VS019-8AF3 OPEN",
                           Diag_Alarm => "07_DOOR"."DOOR =SC00+UC175.VS019-8AF3 IN ALARM");
END_REGION

REGION Network 20: L8 - SC00+UC214.VS019 ([D022] S4008 | =SC00+UC21.EL001/311)
   // Sorter Gate
   RUNG wire#powerrail
      "GATE_SC00+UC214.VS019"(Bypass_For_Commissioning := "00_Commissioning"."n0066-uc21-el001-k30001_SN51", DIAG := TRUE, CH1 := "SAFETY DOOR OPEN =SC00+UC214.VS019-8AF3 (SAFE CH1 =SC00+UC214.VS019)", CH2 := "SAFETY DOOR OPEN =SC00+UC214.VS019-8AF3 (SAFE CH2 =SC00+UC214.VS019)", "Sorter_Running_from MSC" :=, Sorter_Stop_from_Encoder :=, Open_Request :=, Alarm_Filter :=, Sorter_Door := FALSE, ACK_NEC :=, ACK :=, Solenoid =>, EM_Cut => "07_DOOR"."DOOR =SC00+UC214.VS019-8AF3 EM_CUT", EM_Cut_Delay =>, Diag_Open => "07_DOOR"."DOOR =SC00+UC214.VS019-8AF3 OPEN", Diag_Alarm => "07_DOOR"."DOOR =SC00+UC214.VS019-8AF3 IN ALARM")
   END_RUNG
   // the same network as SCL:
   "GATE_SC00+UC214.VS019"(Bypass_For_Commissioning := "00_Commissioning"."n0066-uc21-el001-k30001_SN51",   // "02_Safety_Door"
                           DIAG := TRUE,
                           CH1 := "SAFETY DOOR OPEN =SC00+UC214.VS019-8AF3 (SAFE CH1 =SC00+UC214.VS019)",
                           CH2 := "SAFETY DOOR OPEN =SC00+UC214.VS019-8AF3 (SAFE CH2 =SC00+UC214.VS019)",
                           Sorter_Door := FALSE,
                           EM_Cut => "07_DOOR"."DOOR =SC00+UC214.VS019-8AF3 EM_CUT",
                           Diag_Open => "07_DOOR"."DOOR =SC00+UC214.VS019-8AF3 OPEN",
                           Diag_Alarm => "07_DOOR"."DOOR =SC00+UC214.VS019-8AF3 IN ALARM");
END_REGION

REGION Network 21: L9 - SC00+UC224.VS019 ([D021] S4009 | =SC00+UC22.EL001/311)
   // Sorter Gate
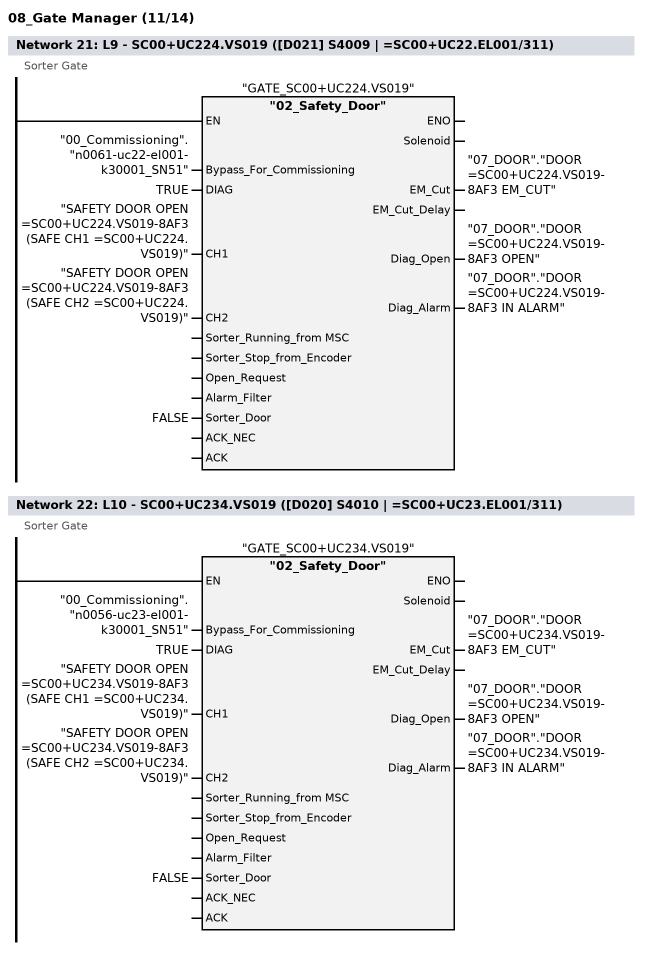
   RUNG wire#powerrail
      "GATE_SC00+UC224.VS019"(Bypass_For_Commissioning := "00_Commissioning"."n0061-uc22-el001-k30001_SN51", DIAG := TRUE, CH1 := "SAFETY DOOR OPEN =SC00+UC224.VS019-8AF3 (SAFE CH1 =SC00+UC224.VS019)", CH2 := "SAFETY DOOR OPEN =SC00+UC224.VS019-8AF3 (SAFE CH2 =SC00+UC224.VS019)", "Sorter_Running_from MSC" :=, Sorter_Stop_from_Encoder :=, Open_Request :=, Alarm_Filter :=, Sorter_Door := FALSE, ACK_NEC :=, ACK :=, Solenoid =>, EM_Cut => "07_DOOR"."DOOR =SC00+UC224.VS019-8AF3 EM_CUT", EM_Cut_Delay =>, Diag_Open => "07_DOOR"."DOOR =SC00+UC224.VS019-8AF3 OPEN", Diag_Alarm => "07_DOOR"."DOOR =SC00+UC224.VS019-8AF3 IN ALARM")
   END_RUNG
   // the same network as SCL:
   "GATE_SC00+UC224.VS019"(Bypass_For_Commissioning := "00_Commissioning"."n0061-uc22-el001-k30001_SN51",   // "02_Safety_Door"
                           DIAG := TRUE,
                           CH1 := "SAFETY DOOR OPEN =SC00+UC224.VS019-8AF3 (SAFE CH1 =SC00+UC224.VS019)",
                           CH2 := "SAFETY DOOR OPEN =SC00+UC224.VS019-8AF3 (SAFE CH2 =SC00+UC224.VS019)",
                           Sorter_Door := FALSE,
                           EM_Cut => "07_DOOR"."DOOR =SC00+UC224.VS019-8AF3 EM_CUT",
                           Diag_Open => "07_DOOR"."DOOR =SC00+UC224.VS019-8AF3 OPEN",
                           Diag_Alarm => "07_DOOR"."DOOR =SC00+UC224.VS019-8AF3 IN ALARM");
END_REGION

REGION Network 22: L10 - SC00+UC234.VS019 ([D020] S4010 | =SC00+UC23.EL001/311)
   // Sorter Gate
   RUNG wire#powerrail
      "GATE_SC00+UC234.VS019"(Bypass_For_Commissioning := "00_Commissioning"."n0056-uc23-el001-k30001_SN51", DIAG := TRUE, CH1 := "SAFETY DOOR OPEN =SC00+UC234.VS019-8AF3 (SAFE CH1 =SC00+UC234.VS019)", CH2 := "SAFETY DOOR OPEN =SC00+UC234.VS019-8AF3 (SAFE CH2 =SC00+UC234.VS019)", "Sorter_Running_from MSC" :=, Sorter_Stop_from_Encoder :=, Open_Request :=, Alarm_Filter :=, Sorter_Door := FALSE, ACK_NEC :=, ACK :=, Solenoid =>, EM_Cut => "07_DOOR"."DOOR =SC00+UC234.VS019-8AF3 EM_CUT", EM_Cut_Delay =>, Diag_Open => "07_DOOR"."DOOR =SC00+UC234.VS019-8AF3 OPEN", Diag_Alarm => "07_DOOR"."DOOR =SC00+UC234.VS019-8AF3 IN ALARM")
   END_RUNG
   // the same network as SCL:
   "GATE_SC00+UC234.VS019"(Bypass_For_Commissioning := "00_Commissioning"."n0056-uc23-el001-k30001_SN51",   // "02_Safety_Door"
                           DIAG := TRUE,
                           CH1 := "SAFETY DOOR OPEN =SC00+UC234.VS019-8AF3 (SAFE CH1 =SC00+UC234.VS019)",
                           CH2 := "SAFETY DOOR OPEN =SC00+UC234.VS019-8AF3 (SAFE CH2 =SC00+UC234.VS019)",
                           Sorter_Door := FALSE,
                           EM_Cut => "07_DOOR"."DOOR =SC00+UC234.VS019-8AF3 EM_CUT",
                           Diag_Open => "07_DOOR"."DOOR =SC00+UC234.VS019-8AF3 OPEN",
                           Diag_Alarm => "07_DOOR"."DOOR =SC00+UC234.VS019-8AF3 IN ALARM");
END_REGION

REGION Network 23: L11 - SC00+UC244.VS019 ([D019] S4011 | =SC00+UC24.EL001/311)
   // Sorter Gate
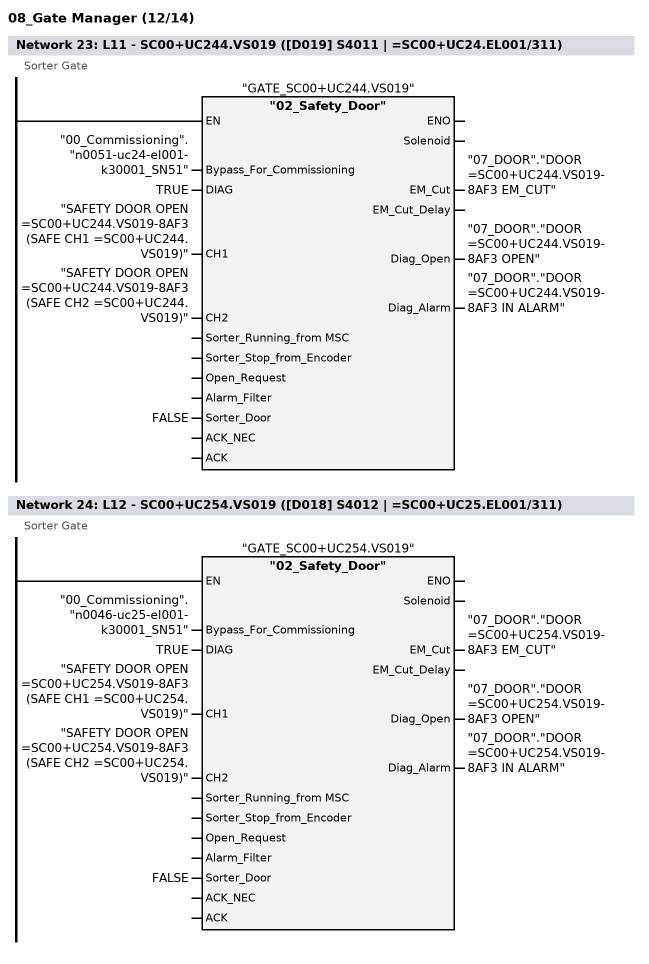
   RUNG wire#powerrail
      "GATE_SC00+UC244.VS019"(Bypass_For_Commissioning := "00_Commissioning"."n0051-uc24-el001-k30001_SN51", DIAG := TRUE, CH1 := "SAFETY DOOR OPEN =SC00+UC244.VS019-8AF3 (SAFE CH1 =SC00+UC244.VS019)", CH2 := "SAFETY DOOR OPEN =SC00+UC244.VS019-8AF3 (SAFE CH2 =SC00+UC244.VS019)", "Sorter_Running_from MSC" :=, Sorter_Stop_from_Encoder :=, Open_Request :=, Alarm_Filter :=, Sorter_Door := FALSE, ACK_NEC :=, ACK :=, Solenoid =>, EM_Cut => "07_DOOR"."DOOR =SC00+UC244.VS019-8AF3 EM_CUT", EM_Cut_Delay =>, Diag_Open => "07_DOOR"."DOOR =SC00+UC244.VS019-8AF3 OPEN", Diag_Alarm => "07_DOOR"."DOOR =SC00+UC244.VS019-8AF3 IN ALARM")
   END_RUNG
   // the same network as SCL:
   "GATE_SC00+UC244.VS019"(Bypass_For_Commissioning := "00_Commissioning"."n0051-uc24-el001-k30001_SN51",   // "02_Safety_Door"
                           DIAG := TRUE,
                           CH1 := "SAFETY DOOR OPEN =SC00+UC244.VS019-8AF3 (SAFE CH1 =SC00+UC244.VS019)",
                           CH2 := "SAFETY DOOR OPEN =SC00+UC244.VS019-8AF3 (SAFE CH2 =SC00+UC244.VS019)",
                           Sorter_Door := FALSE,
                           EM_Cut => "07_DOOR"."DOOR =SC00+UC244.VS019-8AF3 EM_CUT",
                           Diag_Open => "07_DOOR"."DOOR =SC00+UC244.VS019-8AF3 OPEN",
                           Diag_Alarm => "07_DOOR"."DOOR =SC00+UC244.VS019-8AF3 IN ALARM");
END_REGION

REGION Network 24: L12 - SC00+UC254.VS019 ([D018] S4012 | =SC00+UC25.EL001/311)
   // Sorter Gate
   RUNG wire#powerrail
      "GATE_SC00+UC254.VS019"(Bypass_For_Commissioning := "00_Commissioning"."n0046-uc25-el001-k30001_SN51", DIAG := TRUE, CH1 := "SAFETY DOOR OPEN =SC00+UC254.VS019-8AF3 (SAFE CH1 =SC00+UC254.VS019)", CH2 := "SAFETY DOOR OPEN =SC00+UC254.VS019-8AF3 (SAFE CH2 =SC00+UC254.VS019)", "Sorter_Running_from MSC" :=, Sorter_Stop_from_Encoder :=, Open_Request :=, Alarm_Filter :=, Sorter_Door := FALSE, ACK_NEC :=, ACK :=, Solenoid =>, EM_Cut => "07_DOOR"."DOOR =SC00+UC254.VS019-8AF3 EM_CUT", EM_Cut_Delay =>, Diag_Open => "07_DOOR"."DOOR =SC00+UC254.VS019-8AF3 OPEN", Diag_Alarm => "07_DOOR"."DOOR =SC00+UC254.VS019-8AF3 IN ALARM")
   END_RUNG
   // the same network as SCL:
   "GATE_SC00+UC254.VS019"(Bypass_For_Commissioning := "00_Commissioning"."n0046-uc25-el001-k30001_SN51",   // "02_Safety_Door"
                           DIAG := TRUE,
                           CH1 := "SAFETY DOOR OPEN =SC00+UC254.VS019-8AF3 (SAFE CH1 =SC00+UC254.VS019)",
                           CH2 := "SAFETY DOOR OPEN =SC00+UC254.VS019-8AF3 (SAFE CH2 =SC00+UC254.VS019)",
                           Sorter_Door := FALSE,
                           EM_Cut => "07_DOOR"."DOOR =SC00+UC254.VS019-8AF3 EM_CUT",
                           Diag_Open => "07_DOOR"."DOOR =SC00+UC254.VS019-8AF3 OPEN",
                           Diag_Alarm => "07_DOOR"."DOOR =SC00+UC254.VS019-8AF3 IN ALARM");
END_REGION

REGION Network 25: L13 - SC00+UC264.VS019 ([D016] S4013 | =SC00+UC26.EL001/311)
   // Sorter Gate
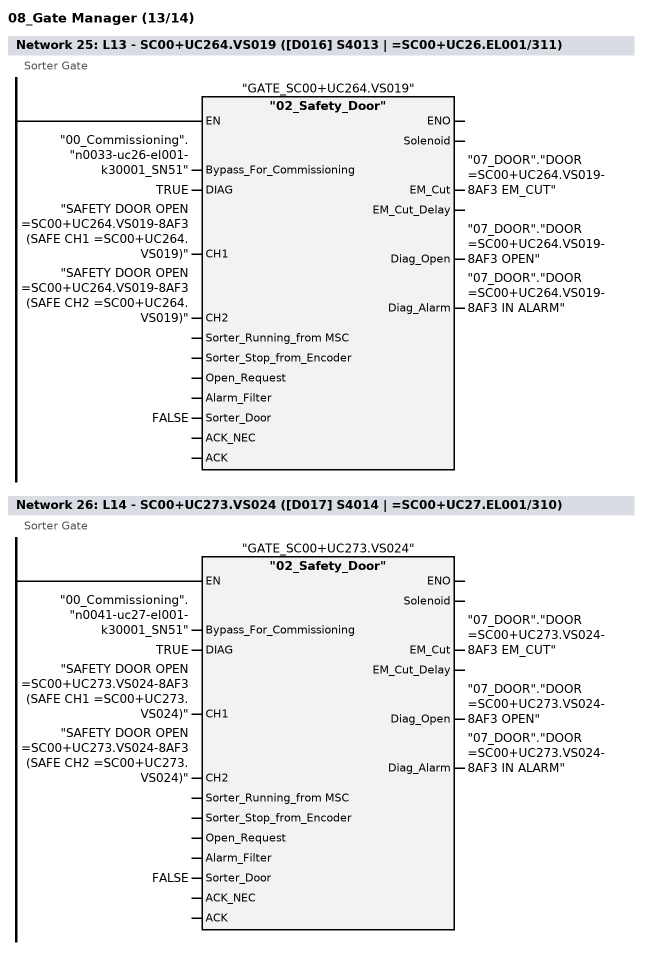
   RUNG wire#powerrail
      "GATE_SC00+UC264.VS019"(Bypass_For_Commissioning := "00_Commissioning"."n0033-uc26-el001-k30001_SN51", DIAG := TRUE, CH1 := "SAFETY DOOR OPEN =SC00+UC264.VS019-8AF3 (SAFE CH1 =SC00+UC264.VS019)", CH2 := "SAFETY DOOR OPEN =SC00+UC264.VS019-8AF3 (SAFE CH2 =SC00+UC264.VS019)", "Sorter_Running_from MSC" :=, Sorter_Stop_from_Encoder :=, Open_Request :=, Alarm_Filter :=, Sorter_Door := FALSE, ACK_NEC :=, ACK :=, Solenoid =>, EM_Cut => "07_DOOR"."DOOR =SC00+UC264.VS019-8AF3 EM_CUT", EM_Cut_Delay =>, Diag_Open => "07_DOOR"."DOOR =SC00+UC264.VS019-8AF3 OPEN", Diag_Alarm => "07_DOOR"."DOOR =SC00+UC264.VS019-8AF3 IN ALARM")
   END_RUNG
   // the same network as SCL:
   "GATE_SC00+UC264.VS019"(Bypass_For_Commissioning := "00_Commissioning"."n0033-uc26-el001-k30001_SN51",   // "02_Safety_Door"
                           DIAG := TRUE,
                           CH1 := "SAFETY DOOR OPEN =SC00+UC264.VS019-8AF3 (SAFE CH1 =SC00+UC264.VS019)",
                           CH2 := "SAFETY DOOR OPEN =SC00+UC264.VS019-8AF3 (SAFE CH2 =SC00+UC264.VS019)",
                           Sorter_Door := FALSE,
                           EM_Cut => "07_DOOR"."DOOR =SC00+UC264.VS019-8AF3 EM_CUT",
                           Diag_Open => "07_DOOR"."DOOR =SC00+UC264.VS019-8AF3 OPEN",
                           Diag_Alarm => "07_DOOR"."DOOR =SC00+UC264.VS019-8AF3 IN ALARM");
END_REGION

REGION Network 26: L14 - SC00+UC273.VS024 ([D017] S4014 | =SC00+UC27.EL001/310)
   // Sorter Gate
   RUNG wire#powerrail
      "GATE_SC00+UC273.VS024"(Bypass_For_Commissioning := "00_Commissioning"."n0041-uc27-el001-k30001_SN51", DIAG := TRUE, CH1 := "SAFETY DOOR OPEN =SC00+UC273.VS024-8AF3 (SAFE CH1 =SC00+UC273.VS024)", CH2 := "SAFETY DOOR OPEN =SC00+UC273.VS024-8AF3 (SAFE CH2 =SC00+UC273.VS024)", "Sorter_Running_from MSC" :=, Sorter_Stop_from_Encoder :=, Open_Request :=, Alarm_Filter :=, Sorter_Door := FALSE, ACK_NEC :=, ACK :=, Solenoid =>, EM_Cut => "07_DOOR"."DOOR =SC00+UC273.VS024-8AF3 EM_CUT", EM_Cut_Delay =>, Diag_Open => "07_DOOR"."DOOR =SC00+UC273.VS024-8AF3 OPEN", Diag_Alarm => "07_DOOR"."DOOR =SC00+UC273.VS024-8AF3 IN ALARM")
   END_RUNG
   // the same network as SCL:
   "GATE_SC00+UC273.VS024"(Bypass_For_Commissioning := "00_Commissioning"."n0041-uc27-el001-k30001_SN51",   // "02_Safety_Door"
                           DIAG := TRUE,
                           CH1 := "SAFETY DOOR OPEN =SC00+UC273.VS024-8AF3 (SAFE CH1 =SC00+UC273.VS024)",
                           CH2 := "SAFETY DOOR OPEN =SC00+UC273.VS024-8AF3 (SAFE CH2 =SC00+UC273.VS024)",
                           Sorter_Door := FALSE,
                           EM_Cut => "07_DOOR"."DOOR =SC00+UC273.VS024-8AF3 EM_CUT",
                           Diag_Open => "07_DOOR"."DOOR =SC00+UC273.VS024-8AF3 OPEN",
                           Diag_Alarm => "07_DOOR"."DOOR =SC00+UC273.VS024-8AF3 IN ALARM");
END_REGION

REGION Network 27: L15 - SF00+UF511.VS015 ([D023] S4029 | =SF00+UF51.EL001/310)
   // Sorter Gate
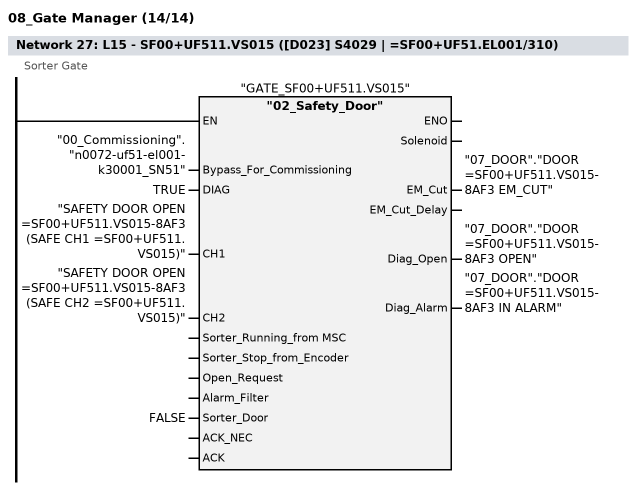
   RUNG wire#powerrail
      "GATE_SF00+UF511.VS015"(Bypass_For_Commissioning := "00_Commissioning"."n0072-uf51-el001-k30001_SN51", DIAG := TRUE, CH1 := "SAFETY DOOR OPEN =SF00+UF511.VS015-8AF3 (SAFE CH1 =SF00+UF511.VS015)", CH2 := "SAFETY DOOR OPEN =SF00+UF511.VS015-8AF3 (SAFE CH2 =SF00+UF511.VS015)", "Sorter_Running_from MSC" :=, Sorter_Stop_from_Encoder :=, Open_Request :=, Alarm_Filter :=, Sorter_Door := FALSE, ACK_NEC :=, ACK :=, Solenoid =>, EM_Cut => "07_DOOR"."DOOR =SF00+UF511.VS015-8AF3 EM_CUT", EM_Cut_Delay =>, Diag_Open => "07_DOOR"."DOOR =SF00+UF511.VS015-8AF3 OPEN", Diag_Alarm => "07_DOOR"."DOOR =SF00+UF511.VS015-8AF3 IN ALARM")
   END_RUNG
   // the same network as SCL:
   "GATE_SF00+UF511.VS015"(Bypass_For_Commissioning := "00_Commissioning"."n0072-uf51-el001-k30001_SN51",   // "02_Safety_Door"
                           DIAG := TRUE,
                           CH1 := "SAFETY DOOR OPEN =SF00+UF511.VS015-8AF3 (SAFE CH1 =SF00+UF511.VS015)",
                           CH2 := "SAFETY DOOR OPEN =SF00+UF511.VS015-8AF3 (SAFE CH2 =SF00+UF511.VS015)",
                           Sorter_Door := FALSE,
                           EM_Cut => "07_DOOR"."DOOR =SF00+UF511.VS015-8AF3 EM_CUT",
                           Diag_Open => "07_DOOR"."DOOR =SF00+UF511.VS015-8AF3 OPEN",
                           Diag_Alarm => "07_DOOR"."DOOR =SF00+UF511.VS015-8AF3 IN ALARM");
END_REGION
END_FUNCTION
